Fanuc KAREL source: kb00051.KL

-- PROVISIONAL review KL for V1013-1; original PC SHA256 2350a1f68f73269a1cd3ef171766a07630ae456a8012564bf5be2baa293cdd72
-- Incomplete behavior may be omitted. Consult companion uncertainty JSON. Do not deploy.
PROGRAM KB00051
%NOLOCKGROUP
VAR
  P1 : INTEGER
  P2 : INTEGER
-- UNRESOLVED_DECL RESULT type=000199
BEGIN
  -- UNRESOLVED_PC offsets 5-12; opcodes 9D,23
  -- UNRESOLVED_PC offsets 17-24; opcodes 9D,23
  -- UNRESOLVED_PC offsets 29-58; opcodes 27,22,22,27,9D,76,7E,4A
  -- UNRESOLVED_PC offsets 63-67; opcodes 7F
END KB00051
